(* IEC 61131-3 sources: CodesysTest/alpha/export/FBs/Components/FB_MurrK50/Advanced Mode, 5 files *)

(* ---- K50AnimationDirection.dut.st ---- *)
(*#-#-#-#-#-#-#-#-#-#---Declaration---#-#-#-#-#-#-#-#-#-#-#-#-#*)

{attribute 'qualified_only'}
{attribute 'strict'}
TYPE K50AnimationDirection :
(
	CCW := 0,
	CW := 1
);
END_TYPE

(* ---- K50AnimationPatterns.dut.st ---- *)
(*#-#-#-#-#-#-#-#-#-#---Declaration---#-#-#-#-#-#-#-#-#-#-#-#-#*)

{attribute 'qualified_only'}
{attribute 'strict'}
TYPE K50AnimationPatterns :
(
	 Flash := 0,
     Strobe := 1,
	 ThreePulse := 2,
	 SOS := 3,
	 Random := 4
);
END_TYPE

(* ---- K50AnimationTypes.dut.st ---- *)
(*#-#-#-#-#-#-#-#-#-#---Declaration---#-#-#-#-#-#-#-#-#-#-#-#-#*)

{attribute 'qualified_only'}
{attribute 'strict'}
TYPE K50AnimationTypes :
(
	Off := 0,
    Steady := 1,
	Flash := 2,
	TwoColorFlash := 3,
	fiftyfifty := 4,
	fiftyfiftyRotate := 5,
	Chase := 6,
	IntensitySweep := 7,
	ColorSweep := 8
);
END_TYPE

(* ---- K50Colors.dut.st ---- *)
(*#-#-#-#-#-#-#-#-#-#---Declaration---#-#-#-#-#-#-#-#-#-#-#-#-#*)

{attribute 'qualified_only'}
{attribute 'strict'}
TYPE K50Colors :
(
	Green := 0,
    Red := 1,
    Orange := 2,
    Amber := 3,
    Yellow := 4,
    LimeGreen := 5,
    SpringGreen := 6,
    Cyan := 7,
    SkyBlue := 8,
    Blue := 9,
    Violet := 10,
    Magenta := 11,
    Rose := 12,
    White := 13,
    Custom1 := 14,
    Custom2 := 15
) BYTE ;
END_TYPE

(* ---- FB_MurrK50_AdvancedMode.pou.st ---- *)
(*#-#-#-#-#-#-#-#-#-#---Declaration---#-#-#-#-#-#-#-#-#-#-#-#-#*)

FUNCTION_BLOCK FB_MurrK50_AdvancedMode
VAR_INPUT
	IOLinkData : POINTER TO ARRAY[0..9] OF BYTE;
	baggerReady : BOOL;
	baggerFaulted : BOOL;
	baggerInCycle : BOOL;
	baggerExternalInhibited : BOOL;
END_VAR
VAR
	_IOLinkStateOutput : BYTE;
	_IOLinkData : ARRAY[0..9] OF BYTE;
	_baggerNotReadyProfile : K50OutputProfile :=
		(animationType := K50AnimationTypes.Off,
  dynamicSequenceValue := 0);

  	_baggerReadyProfile : K50OutputProfile :=
			 (colorOne := K50Colors.Green,
              colorTwo := K50Colors.Green,
         animationType := K50AnimationTypes.Steady,
  dynamicSequenceValue := 0);

  	_baggerInCycleProfile : K50OutputProfile :=
			 (colorOne := K50Colors.Green,
              colorTwo := K50Colors.White,
         animationType := K50AnimationTypes.fiftyfiftyRotate,
        animationSpeed := K50AnimationSpeeds.Medium,
    animationDirection := K50AnimationDirection.CCW,
     animationPatterns := K50AnimationPatterns.Flash,
  dynamicSequenceValue := 0);

    	_baggerInhibitedProfile : K50OutputProfile :=
			 (colorOne := K50Colors.Yellow,
              colorTwo := K50Colors.White,
         animationType := K50AnimationTypes.fiftyfiftyRotate,
        animationSpeed := K50AnimationSpeeds.Medium,
    animationDirection := K50AnimationDirection.CCW,
     animationPatterns := K50AnimationPatterns.Flash,
  dynamicSequenceValue := 0);

  	_baggerFaultedProfile : K50OutputProfile :=
			 (colorOne := K50Colors.Red,
              colorTwo := K50Colors.Red,
         animationType := K50AnimationTypes.Flash,
        animationSpeed := K50AnimationSpeeds.Medium,
    animationDirection := K50AnimationDirection.CCW,
     animationPatterns := K50AnimationPatterns.Flash,
  dynamicSequenceValue := 0);

  	_profiles : ARRAY[0..4] OF K50OutputProfile := [_baggerNotReadyProfile,
													_baggerReadyProfile,
													_baggerInCycleProfile,
													_baggerInhibitedProfile,
													_baggerFaultedProfile];
END_VAR
(*#-#-#-#-#-#-#-#-#-#---Implementation---#-#-#-#-#-#-#-#-#-#-#-#-#*)

//
//  FB_MurrK50_AdvancedMode
//  FBs/FB_MurrK50/Advanced Mode/FB_MurrK50_AdvancedMode
//
//  Created by Evan Ische on 6/17/2021.
//  Copyright (C) 2021 Sharp Packaging Systems By Pregis. All rights reserved.
//

//
_IOLinkStateOutput := 0;
IF baggerReady THEN
	_IOLinkStateOutput := 1;
END_IF
IF baggerInCycle THEN
	_IOLinkStateOutput := 2;
END_IF
IF baggerExternalInhibited THEN
	_IOLinkStateOutput := 3;
END_IF
IF baggerFaulted THEN
	_IOLinkStateOutput := 4;
END_IF

// Write The Selected Profiles Data To The Correct IO-Link Bytes
_IOLinkData[0] := _profiles[_IOLinkStateOutput].colorTwo;
_IOLinkData[1] := _profiles[_IOLinkStateOutput].colorOne;
_IOLinkData[3] := _profiles[_IOLinkStateOutput].dynamicSequenceValue;
_IOLinkData[6].0 := _profiles[_IOLinkStateOutput].animationSpeed.0;
_IOLinkData[6].1 := _profiles[_IOLinkStateOutput].animationSpeed.1;
_IOLinkData[6].2 := _profiles[_IOLinkStateOutput].vibrationFeedback.0;
_IOLinkData[6].3 := _profiles[_IOLinkStateOutput].vibrationFeedback.1;
_IOLinkData[7].0 := _profiles[_IOLinkStateOutput].animationType.0;
_IOLinkData[7].1 := _profiles[_IOLinkStateOutput].animationType.1;
_IOLinkData[7].2 := _profiles[_IOLinkStateOutput].animationType.2;
_IOLinkData[7].3 := _profiles[_IOLinkStateOutput].animationType.3;
_IOLinkData[7].4 := _profiles[_IOLinkStateOutput].animationDirection.0;
_IOLinkData[7].5 := _profiles[_IOLinkStateOutput].animationPatterns.0;
_IOLinkData[7].6 := _profiles[_IOLinkStateOutput].animationPatterns.1;
_IOLinkData[7].7 := _profiles[_IOLinkStateOutput].animationPatterns.2;
IOLinkData^ := _IOLinkData;
